FUNCTION_BLOCK FB_Fifo
VAR CONSTANT
	NoOfEntries: INT := 100;
END_VAR
VAR_INPUT
END_VAR
VAR_OUTPUT
	bDataInBuffer: BOOL;
	bBufferFull: BOOL;
	MaxBuffer : INT;
END_VAR
VAR
	Buffer : ARRAY[0..NoOfEntries] OF ST_streamOutputs;
	init: BOOL := true;
	index: INT;
END_VAR


IF init THEN
	index := 0;
	MaxBuffer := 0;
	init := FALSE;
END_IF

bDataInBuffer := index > 0;
bBufferFull := index >= NoOfEntries;


IF index > MaxBuffer THEN
	Maxbuffer := index;
END_IF

METHOD M_AddEntry : BOOL
VAR_INPUT
	cycleNo : UDINT;
	on : BOOL;

END_VAR
VAR_OUTPUT
	bError: BOOL;
END_VAR
VAR
		stEntry : ST_streamOutputs;
END_VAR

IF (index < NoOfEntries) THEN
	stEntry.cycleNo := cycleNo;
	stEntry.on := on;
	
	Buffer[index] := stEntry;
	index := index + 1;
	M_AddEntry :=TRUE;
	bError := FALSE;
ELSE
	bError := TRUE;	
END_IF
END_METHOD

METHOD M_init : BOOL
VAR_INPUT
END_VAR
init := true;
END_METHOD

METHOD M_RemoveEntry : ST_streamOutputs
VAR_INPUT
END_VAR

VAR
	n: INT;
END_VAR


IF (index > 0) THEN
	M_RemoveEntry := Buffer[0];

	MEMCPY(destAddr:= ADR(Buffer[0]), srcAddr:=ADR(Buffer[1]), n:=(SIZEOF(Buffer)-SIZEOF(Buffer[1])));
	MEMSET(ADR(Buffer[index]), 0, SIZEOF(Buffer[index]));
	index := index -1;

END_IF
END_METHOD

END_FUNCTION_BLOCK

(* stored: Version 1.1.0.1, ProductVersion 3.1.4024.9
   POU FB_Fifo: Id {dd90151b-8b71-44b8-8e80-521f5f62c591}, SpecialFunc None
   Method M_AddEntry: Id {59eb4391-e9d5-4878-afa9-cbca16d92f55}
   Method M_init: Id {0dce51b4-2438-4688-8c68-1850a893a463}
   Method M_RemoveEntry: Id {d5d765b9-1bec-49ef-8bf7-6d44a13fdb27} *)
